// TIA Portal V20 export
VAR_GLOBAL   // PLC tag table "ConvConstantPackedLine"
END_VAR
VAR_GLOBAL CONSTANT   // user constants
   minPackedLine : Int := 3001;
   maxPackedLine : Int := 3040;
   "G1.1.1" : Int := 3001;   // G1.1.1
   "G1.1.2" : Int := 3002;   // G1.1.2
   "G1.1.3" : Int := 3003;   // G1.1.3
   "G1.1.4" : Int := 3004;   // G1.1.4
   "G1.1.5" : Int := 3005;   // G1.1.5
   "G1.1.6" : Int := 3006;   // G1.1.6
   "G1.1.7" : Int := 3007;   // G1.1.7
   "G1.1.8" : Int := 3008;   // G1.1.8
   "G1.1.9" : Int := 3009;   // G1.1.9
   "G1.1.10" : Int := 3010;   // G1.1.10
   "G1.1.11" : Int := 3011;   // G1.1.11
   "G1.1.12" : Int := 3012;   // G1.1.12
   "G1.1.13" : Int := 3013;   // G1.1.13
   "G1.1.14" : Int := 3014;   // G1.1.14
   "G1.1.15" : Int := 3015;   // G1.1.15
   "G1.1.16" : Int := 3016;   // G1.1.16
   "G1.1.17" : Int := 3017;   // G1.1.17
   "G1.1.18" : Int := 3018;   // G1.1.18
   "G1.1.19" : Int := 3019;   // G1.1.19
   "G1.2.1" : Int := 3020;   // G1.2.1
   "G1.2.2" : Int := 3021;   // G1.2.2
   "G1.3.1" : Int := 3022;   // G1.3.1
   "G1.4.1" : Int := 3023;   // G1.4.1
   "G1.4.2" : Int := 3024;   // G1.4.2
   "G1.4.3" : Int := 3025;   // G1.4.3
   "G1.4.4" : Int := 3026;   // G1.4.4
   "G1.4.5" : Int := 3027;   // G1.4.5
   "G1.4.6" : Int := 3028;   // G1.4.6
   "G1.5.1" : Int := 3029;   // G1.5.1
   "G1.5.2" : Int := 3030;   // G1.5.2
   "G1.5.3" : Int := 3031;   // G1.5.3
   "G1.5.4" : Int := 3032;   // G1.5.4
   "G1.5.5" : Int := 3033;   // G1.5.5
   "G1.5.6" : Int := 3034;   // G1.5.6
   "G1.6.1" : Int := 3035;   // G1.6.1
   "G1.6.2" : Int := 3036;   // G1.6.2
   "G1.7.1" : Int := 3037;   // G1.7.1
   "G1.7.2" : Int := 3038;   // G1.7.2
   "G1.7.3" : Int := 3039;   // G1.7.3
   "G1.7.4" : Int := 3040;   // G1.7.4
END_VAR
